// TIA Portal V20 export
// export: Created 2026-07-17T22:20:22.6742411Z, ExportSetting WithDefaults, DisplayName Totally Integrated Automation Portal, DisplayVersion V20 Update 5, DisplayName TIA Portal Openness, DisplayVersion V20 Update 4, DisplayName TIA Portal Version Control Interface, DisplayVersion V20 Update 5, DisplayName SINAMICS Startdrive Advanced, DisplayVersion V20, DisplayName SINAMICS DCC, DisplayVersion V20, DisplayName SINAMICS Startdrive G130, G150, S120, S150, SINAMICS MV, G220, S200, S210, DisplayVersion V20, DisplayName SINAMICS Startdrive G110M, G120, G120C, G120D, G120P, G115D, DisplayVersion V20, DisplayName STEP 7 Professional, DisplayVersion V20 Update 5, DisplayName STEP 7 Safety, DisplayVersion V20 Update 2, DisplayName WinCC Basic/Comfort/Advanced, DisplayVersion V20 Update 5, DisplayName WinCC Unified, DisplayVersion V20 Update 5
ORGANIZATION_BLOCK "OB100"   // OB100, LAD, Startup
TITLE = Startup Reset
{ S7_Optimized_Access := 'TRUE' }
VERSION : 0.1
// Dedicated startup-reset block (C-124/C-305/C-403), run once by the CPU on every restart (warm or cold), regardless of retentivity - non-retentivity is never relied on to clear state. Forces Step back to idle (C-118/C-119) on every stepped sequencer, clears every S/R-driven and transient-run-state bit named in the fix-wave-1 B-2 finding, and force-resets DB_PLC.Simulation (C-305). Genuine fault latches - iDB_MotorFwdRevSystem_Shredder.IO.FaultActive/FTR/FTS, iDB_PusherControl.IO.Blocked/EndTravelTimeoutFault/ParkedTimeoutFault/BothSwitchesFault, iDB_ShredderSequencer.IO.ShredderBlockedFault/DischargeConveyorTimeoutFault - are deliberately excluded per C-124's carve-out: a fault needing human acknowledgement (FaultReset) still needs it after a power cycle. Closes owner-questions B-2/D-1/Q-01 and doc 06 C-128 (no automatic restart after a stop or power event).
// stored: AutoNumber true, IsIECCheckEnabled false, SetENOAutomatically false
   VAR_INPUT
      LostRetentive : Bool;   // True if retentive data are lost
      LostRTC : Bool;   // True if date and time are lost
   END_VAR
BEGIN

REGION Network 1: Shredder sequencer - force Step idle, clear transient state (C-124)
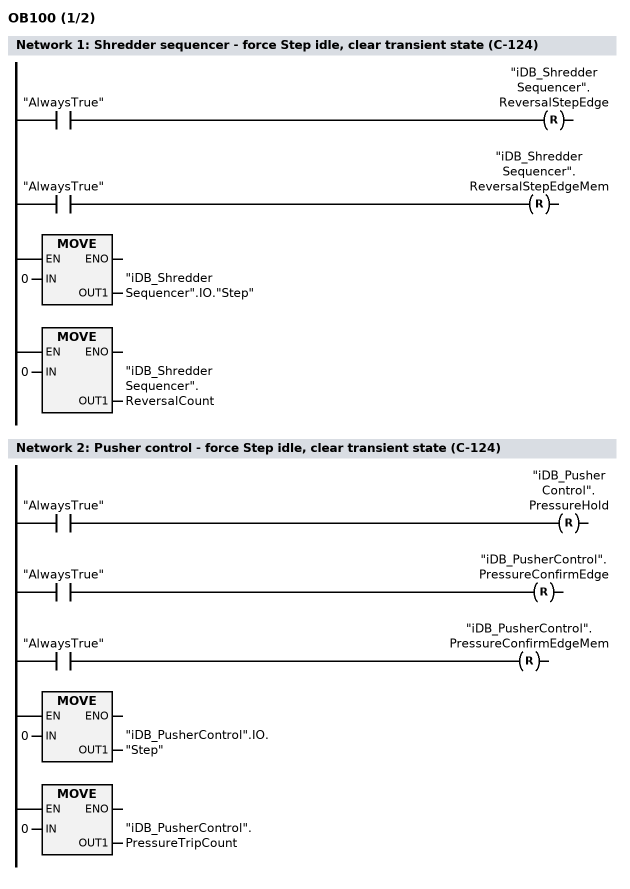
   RUNG wire#powerrail
      Contact( "AlwaysTrue" )
      R_Coil( "iDB_ShredderSequencer".ReversalStepEdge )
   END_RUNG
   RUNG wire#powerrail
      Contact( "AlwaysTrue" )
      R_Coil( "iDB_ShredderSequencer".ReversalStepEdgeMem )
   END_RUNG
   RUNG wire#powerrail
      Move(in := 0, out1 => "iDB_ShredderSequencer".IO."Step")
   END_RUNG
   RUNG wire#powerrail
      Move(in := 0, out1 => "iDB_ShredderSequencer".ReversalCount)
   END_RUNG
   // the same network as SCL:
   IF "AlwaysTrue" THEN
       "iDB_ShredderSequencer".ReversalStepEdge := FALSE;
       "iDB_ShredderSequencer".ReversalStepEdgeMem := FALSE;
   END_IF;
   "iDB_ShredderSequencer".IO."Step" := 0;
   "iDB_ShredderSequencer".ReversalCount := 0;
END_REGION

REGION Network 2: Pusher control - force Step idle, clear transient state (C-124)
   RUNG wire#powerrail
      Contact( "AlwaysTrue" )
      R_Coil( "iDB_PusherControl".PressureHold )
   END_RUNG
   RUNG wire#powerrail
      Contact( "AlwaysTrue" )
      R_Coil( "iDB_PusherControl".PressureConfirmEdge )
   END_RUNG
   RUNG wire#powerrail
      Contact( "AlwaysTrue" )
      R_Coil( "iDB_PusherControl".PressureConfirmEdgeMem )
   END_RUNG
   RUNG wire#powerrail
      Move(in := 0, out1 => "iDB_PusherControl".IO."Step")
   END_RUNG
   RUNG wire#powerrail
      Move(in := 0, out1 => "iDB_PusherControl".PressureTripCount)
   END_RUNG
   // the same network as SCL:
   IF "AlwaysTrue" THEN
       "iDB_PusherControl".PressureHold := FALSE;
       "iDB_PusherControl".PressureConfirmEdge := FALSE;
       "iDB_PusherControl".PressureConfirmEdgeMem := FALSE;
   END_IF;
   "iDB_PusherControl".IO."Step" := 0;
   "iDB_PusherControl".PressureTripCount := 0;
END_REGION

REGION Network 3: Motor FB - clear S/R-driven and transient bits (C-403), fault latches excluded
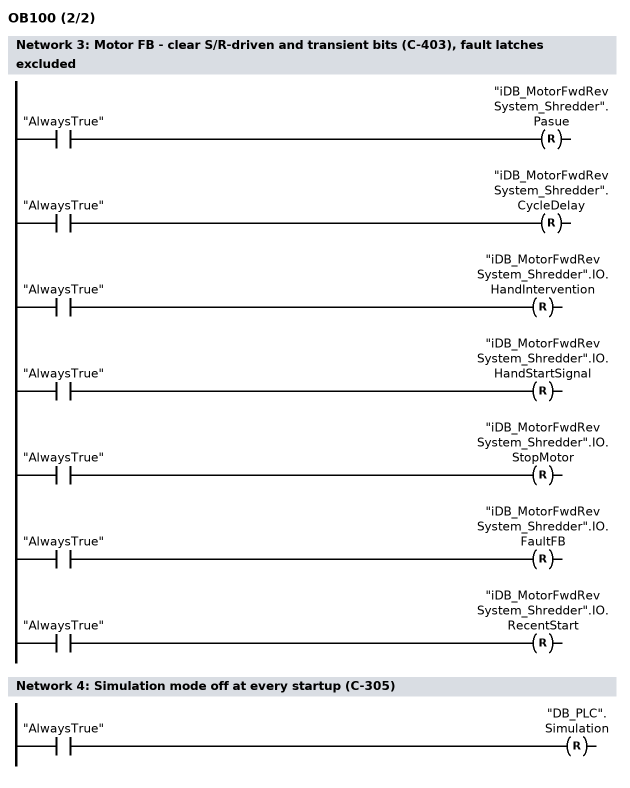
   RUNG wire#powerrail
      Contact( "AlwaysTrue" )
      R_Coil( "iDB_MotorFwdRevSystem_Shredder".Pasue )
   END_RUNG
   RUNG wire#powerrail
      Contact( "AlwaysTrue" )
      R_Coil( "iDB_MotorFwdRevSystem_Shredder".CycleDelay )
   END_RUNG
   RUNG wire#powerrail
      Contact( "AlwaysTrue" )
      R_Coil( "iDB_MotorFwdRevSystem_Shredder".IO.HandIntervention )
   END_RUNG
   RUNG wire#powerrail
      Contact( "AlwaysTrue" )
      R_Coil( "iDB_MotorFwdRevSystem_Shredder".IO.HandStartSignal )
   END_RUNG
   RUNG wire#powerrail
      Contact( "AlwaysTrue" )
      R_Coil( "iDB_MotorFwdRevSystem_Shredder".IO.StopMotor )
   END_RUNG
   RUNG wire#powerrail
      Contact( "AlwaysTrue" )
      R_Coil( "iDB_MotorFwdRevSystem_Shredder".IO.FaultFB )
   END_RUNG
   RUNG wire#powerrail
      Contact( "AlwaysTrue" )
      R_Coil( "iDB_MotorFwdRevSystem_Shredder".IO.RecentStart )
   END_RUNG
   // the same network as SCL:
   IF "AlwaysTrue" THEN
       "iDB_MotorFwdRevSystem_Shredder".Pasue := FALSE;
       "iDB_MotorFwdRevSystem_Shredder".CycleDelay := FALSE;
       "iDB_MotorFwdRevSystem_Shredder".IO.HandIntervention := FALSE;
       "iDB_MotorFwdRevSystem_Shredder".IO.HandStartSignal := FALSE;
       "iDB_MotorFwdRevSystem_Shredder".IO.StopMotor := FALSE;
       "iDB_MotorFwdRevSystem_Shredder".IO.FaultFB := FALSE;
       "iDB_MotorFwdRevSystem_Shredder".IO.RecentStart := FALSE;
   END_IF;
END_REGION

REGION Network 4: Simulation mode off at every startup (C-305)
   RUNG wire#powerrail
      Contact( "AlwaysTrue" )
      R_Coil( "DB_PLC".Simulation )
   END_RUNG
   // the same network as SCL:
   IF "AlwaysTrue" THEN "DB_PLC".Simulation := FALSE; END_IF;
END_REGION
END_ORGANIZATION_BLOCK
